// Mitsubishi GX Works2 project: 7   PLC: FX3U/FX3UC

// task Task_01 (event TRUE, interval 0, priority 31): POU_01

PROGRAM POU_01
VAR
  cnt : INT;
  ii : INT;
  rt1 : R_TRIG;
  ton1 : TON;
END_VAR
IF M8002 THEN
	cnt := -1;
END_IF;

IF M0 THEN
	cnt := 0;
END_IF;

ton1(IN := NOT ton1.Q, PT := T#1s);
rt1(_CLK := ton1.Q AND cnt <> -1);
IF rt1.Q THEN
	cnt := cnt + 1;
	cnt := cnt MOD 4;
END_IF;

IF cnt <> -1 THEN
	FOR ii := 0 TO 3 BY 1 DO
		Z0 := ii;
		Y0Z0 := FALSE;
	END_FOR;
	
	Z0 := cnt;
	Y0Z0 := TRUE;
END_IF;
END_PROGRAM
